{attribute 'qualified_only'}
{attribute 'strict'}
TYPE ST_SF3_2_PSS_ACCESS :
STRUCT
    bSI_PSS_ACCESS : BOOL;
END_STRUCT
END_TYPE

(* stored: Version 1.1.0.1
   DUT ST_SF3_2_PSS_ACCESS: Id {7309269c-1ae7-0ced-290a-1ea86b6a8482} *)
